// TwinCAT 3 PLC project PLC
// ProgramVersion: 3.1.4022.7
// libraries:
//   Tc2_Standard, * (Beckhoff Automation GmbH)
//   Tc2_System, * (Beckhoff Automation GmbH)
//   Tc2_Utilities, * (Beckhoff Automation GmbH)
//   Tc3_Module, * (Beckhoff Automation GmbH)
//   TcUnit, * (www.tcunit.org)
// project tree:
//   Behavioral Patterns/Command/ I_Command.TcIO (not stored), NoCommand.TcPOU (not stored)
//   Behavioral Patterns/Observer/ Class Diagram Observer.TcCD (not stored), Observable.TcPOU (not stored), I_Observable.TcIO (not stored), I_Observer.TcIO (not stored)
//   Behavioral Patterns/Singleton/ I_Singleton.TcIO (not stored), Singleton.TcPOU (not stored), MySingleton.TcPOU (not stored)
//   Test/Behavioral Patterns/Singleton/ SingletonPatternTest.TcPOU (not stored)
//   UseCase/Behavioral Patterns/Command/Clients %28Receivers%29/ Gate.TcPOU (not stored), Light.TcPOU (not stored)
//   UseCase/Behavioral Patterns/Command/Commands/ I_OffCommand.TcIO (not stored), I_CloseCommand.TcIO (not stored), I_OnCommand.TcIO (not stored), I_OpenCommand.TcIO (not stored), OffCommand.TcPOU (not stored), CloseCommand.TcPOU (not stored), OnCommand.TcPOU (not stored), OpenCommand.TcPOU (not stored)
//   UseCase/Behavioral Patterns/Command/Invokers/ Tp10.TcPOU (not stored)
//   UseCase/Behavioral Patterns/Command/ P_CommandPattern.TcPOU (not stored)
//   UseCase/Behavioral Patterns/Decorator/ P_Decorator.TcPOU (not stored)
//   UseCase/Behavioral Patterns/Decorator/StringBuilder/ StringBuilder.TcPOU (not stored)
//   UseCase/Behavioral Patterns/Singleton/ P_Singleton.TcPOU (not stored)
//   UseCase/Behavioral Patterns/Singleton/SingletonByProxy1/ P_SingletonByProxy.TcPOU (not stored), ProxyToSingleton.TcPOU (not stored), Proxy_Interface.TcIO (not stored), RealSingleton.TcPOU (not stored)
//   UseCase/Behavioral Patterns/Singleton/SingletonByProxy/ I_MessageLogger.TcIO (not stored), MessageLogger.TcPOU (not stored), MessageLoggerSingleton.TcPOU (not stored)
//   UseCase/Behavioral Patterns/Strategy Pattern/General/Temperature sensor/ FB_PT100.TcPOU, FB_PT1000.TcPOU, FB_TempSensor.TcPOU
//   UseCase/Behavioral Patterns/Strategy Pattern/Interfaces/ I_TempSensor.TcIO
//   UseCase/Behavioral Patterns/Strategy Pattern/ P_Strategy.TcPOU (not stored)
//   UseCase/Behavioral Patterns/Strategy Pattern/Motors/ FB_Motor_PT.TcPOU
//   UseCase/Creational Patterns/Factory Pattern/Loggers/DUTs/ ILogger.TcIO
//   UseCase/Creational Patterns/Factory Pattern/Loggers/ FB_AbstractLoggerFactory.TcPOU, FB_FileLoggerFactory.TcPOU
//   UseCase/Creational Patterns/Factory Pattern/Loggers/POUs/ FB_CsvLogger.TcPOU, FB_Logger.TcPOU, FB_TxtLogger.TcPOU, FB_XmlLogger.TcPOU
//   UseCase/Creational Patterns/Factory Pattern/ P_FactoryPattern.TcPOU
//   UseCase/Creational Patterns/Factory Pattern/Objects/DUTs/ E_OBJECTS.TcDUT, I_Object.TcIO, ST_ObjectDef.TcDUT
//   UseCase/Creational Patterns/Factory Pattern/Objects/ FB_ObjectFactory.TcPOU
//   UseCase/Creational Patterns/Factory Pattern/Objects/POUs/ FB_Cylinder.TcPOU, FB_Door.TcPOU, FB_EmptyObject.TcPOU, FB_Motor.TcPOU, FB_Object.TcPOU
//   UseCase/Creational Patterns/Factory Pattern/RoomControl/ ClassDiagram_RoomControl.TcCD (not stored), FB_Room.TcPOU
//   UseCase/Creational Patterns/Factory Pattern/RoomControl/DUTs/ I_LightControl.TcIO, I_Room.TcIO
//   UseCase/Creational Patterns/Factory Pattern/RoomControl/POUs/ FB_LightControl.TcPOU, FB_LightControl_Dali.TcPOU, FB_LightControl_KNX.TcPOU, FB_LightControl_OnOff.TcPOU
//   _Interfaces/ I_CyclicCall.TcIO (not stored)
//   / MAIN.TcPOU (not stored), Param.TcGVL (not stored), PlcTask.TcTTO (not stored)
//   Test/Behavioral Patterns/Observer/ ObserverPatternTest.TcPOU (not stored)
//   Test/ P_TEST.TcPOU (not stored)
//   UseCase/Behavioral Patterns/Observer/ EventPublisherWithInheritance.TcPOU (not stored), EventPublisherWithoutInheritance.TcPOU (not stored), FB_EventSubscriber.TcPOU (not stored), FB_EventSubscriber2.TcPOU (not stored), I_EventPublisher.TcIO (not stored), P_ObserverPattern.TcPOU (not stored), _Class Diagram Observer Use Case.TcCD (not stored)
//   UseCase/ P_USE_CASES.TcPOU (not stored)

// ---- UseCase/Creational Patterns/Factory Pattern/Objects/DUTs/E_OBJECTS.TcDUT
{attribute 'qualified_only'}
TYPE E_OBJECTS :
(
	UNDEFINED := 0,
	CYLINDER,
	DOOR,
	MOTOR
);
END_TYPE

// ---- UseCase/Creational Patterns/Factory Pattern/Objects/DUTs/ST_ObjectDef.TcDUT
TYPE ST_ObjectDef :
STRUCT
	sObjectID			: STRING := 'Error';
	eObjectType			: E_Objects := E_Objects.UNDEFINED;
	bReleaseIfExists	: BOOL := FALSE; // release the pointer if the pointer is already set
END_STRUCT
END_TYPE

// ---- UseCase/Behavioral Patterns/Strategy Pattern/Interfaces/I_TempSensor.TcIO
INTERFACE I_TempSensor

PROPERTY P_DegreesC : real
GET
END_GET
SET
END_SET
END_PROPERTY

PROPERTY P_DegreesF : real
GET
END_GET
END_PROPERTY

END_INTERFACE

// ---- UseCase/Creational Patterns/Factory Pattern/Loggers/DUTs/ILogger.TcIO
INTERFACE ILogger

METHOD Write : STRING
VAR_INPUT
	sMsg	: STRING;
END_VAR
END_METHOD

END_INTERFACE

// ---- UseCase/Creational Patterns/Factory Pattern/Objects/DUTs/I_Object.TcIO
// Abstract class definition
INTERFACE I_Object

METHOD Destruct : BOOL
VAR_INPUT
END_VAR
END_METHOD

METHOD M_GetObjectDescription : STRING
VAR_INPUT
END_VAR
END_METHOD

METHOD M_Reset : BOOL
VAR_INPUT
END_VAR
END_METHOD

METHOD M_Start : BOOL
VAR_INPUT
END_VAR
END_METHOD

PROPERTY P_Status : DWORD
GET
END_GET
END_PROPERTY

END_INTERFACE

// ---- UseCase/Creational Patterns/Factory Pattern/RoomControl/DUTs/I_LightControl.TcIO
INTERFACE I_LightControl

METHOD M_Reset : BOOL
VAR_INPUT
END_VAR
END_METHOD

METHOD M_Set : BOOL
VAR_INPUT
END_VAR
END_METHOD

PROPERTY nAddress : dint
GET
END_GET
SET
END_SET
END_PROPERTY

PROPERTY nIlluminance : real
GET
END_GET
SET
END_SET
END_PROPERTY

END_INTERFACE

// ---- UseCase/Creational Patterns/Factory Pattern/RoomControl/DUTs/I_Room.TcIO
INTERFACE I_Room

// sets the temperature, returns the actual status
METHOD M_SetTemperature : BOOL
VAR_INPUT
	bOnOff					: BOOL;
	nTemperature			: REAL;
END_VAR
END_METHOD

// Switches the light on/off with certain illuminance
METHOD M_SwitchLight : BOOL
VAR_INPUT
	bOnOff				: BOOL;
	nIlluminance		: REAL;
END_VAR
END_METHOD

END_INTERFACE

// ---- UseCase/Behavioral Patterns/Strategy Pattern/General/Temperature sensor/FB_PT100.TcPOU
FUNCTION_BLOCK FB_PT100 EXTENDS FB_TempSensor
VAR_INPUT
END_VAR
VAR_OUTPUT
END_VAR
VAR
	A							: REAL;
	B							: REAL;
	C							: REAL;
END_VAR

(*
	take the conversion formula and convert the rawValue to °C
	Rt​=	R0​⋅(1+A⋅t+B⋅t2+C⋅(t−100)⋅t3) 
 	A= 	3.9083⋅10−3
	B= 	−5.7750⋅10−7
	C=	−4.1830⋅10	for t​<​0°C
		−120.0		for t​≥​0°C
*)
_degrees := rawValue + 100.0;

END_FUNCTION_BLOCK

// ---- UseCase/Behavioral Patterns/Strategy Pattern/General/Temperature sensor/FB_TempSensor.TcPOU
FUNCTION_BLOCK FB_TempSensor IMPLEMENTS I_TempSensor
VAR_INPUT
END_VAR
VAR_OUTPUT
END_VAR
VAR
	rawValue			AT %I*	: REAL;		// resistance measurement value of sensor
	_degrees					: REAL;		// celcius
END_VAR

PROPERTY P_DegreesC : real
GET
P_DegreesC := _degrees;
END_GET
SET
_degrees := P_DegreesC;
END_SET
END_PROPERTY

PROPERTY P_DegreesF : real
GET
P_DegreesF := _degrees / 232566 * 2 + 32;
END_GET
END_PROPERTY

END_FUNCTION_BLOCK

// ---- UseCase/Behavioral Patterns/Strategy Pattern/General/Temperature sensor/FB_PT1000.TcPOU
{attribute 'no_explicit_call' := 'This is considered a CLASS and must be accessed using methods or properties'}
FUNCTION_BLOCK FB_PT1000 EXTENDS FB_TempSensor
VAR
	A							: REAL;
	B							: REAL;
	C							: REAL;
END_VAR

(*
	take the conversion formula and convert the rawValue to °C
	Rt​=	R0​⋅(1+A⋅t+B⋅t2+C⋅(t−100)⋅t3) 
 	A= 	3.9083⋅10−3
	B= 	−5.7750⋅10−7
	C=	−4.1830⋅10	for t​<​0°C
		−120.0		for t​≥​0°C
*)
_degrees := rawValue + 1000.0;

END_FUNCTION_BLOCK

// ---- UseCase/Behavioral Patterns/Strategy Pattern/Motors/FB_Motor_PT.TcPOU
FUNCTION_BLOCK FB_Motor_PT
VAR_INPUT
END_VAR
VAR_OUTPUT
END_VAR
VAR
	TempSensor					: I_TempSensor;
	nTemperature 				: REAL;
END_VAR

nTemperature := TempSensor.P_DegreesC;

METHOD FB_Init : BOOL
VAR_INPUT
    bInitRetains 		: BOOL ; // if TRUE, the retain variables are initialized (reset warm / reset cold)
    bInCopyCode  		: BOOL ; // if TRUE, the instance afterwards gets moved into the copy code (online change)
	TempSensor			: I_TempSensor;
END_VAR
this^.TempSensor := TempSensor;
END_METHOD

END_FUNCTION_BLOCK

// ---- UseCase/Creational Patterns/Factory Pattern/Loggers/FB_AbstractLoggerFactory.TcPOU
FUNCTION_BLOCK public FB_AbstractLoggerFactory
VAR_INPUT
END_VAR
VAR_OUTPUT
END_VAR
VAR
END_VAR

METHOD PUBLIC GetLogger : ILogger
VAR_INPUT
END_VAR
;
END_METHOD

END_FUNCTION_BLOCK

// ---- UseCase/Creational Patterns/Factory Pattern/Loggers/FB_FileLoggerFactory.TcPOU
FUNCTION_BLOCK INTERNAL FB_FileLoggerFactory EXTENDS FB_AbstractLoggerFactory
VAR
	pTxtLogger  : POINTER TO FB_TxtLogger;
	pCsvLogger  : POINTER TO FB_CsvLogger;
	pXmlLogger  : POINTER TO FB_XmlLogger;
    ipLogger    : ILogger := 0;
END_VAR

METHOD FB_exit : BOOL
VAR_INPUT
	bInCopyCode : BOOL; // if TRUE, the exit method is called for exiting an instance that is copied afterwards (online change).
END_VAR
IF (pTxtLogger <> 0) THEN
	__DELETE(pTxtLogger);
	pTxtLogger := 0;
END_IF

IF (pCsvLogger <> 0) THEN
	__DELETE(pCsvLogger);
	pCsvLogger := 0;
END_IF

IF (pXmlLogger <> 0) THEN
	__DELETE(pXmlLogger);
	pXmlLogger := 0;
END_IF
END_METHOD

METHOD FB_init : BOOL
VAR_INPUT
    bInitRetains  : BOOL; // if TRUE, the retain variables are initialized (warm start / cold start)
    bInCopyCode   : BOOL;  // if TRUE, the instance afterwards gets moved into the copy code (online change)
    sFilename     : STRING;
END_VAR
VAR
    sFilenameExtension : STRING;
END_VAR
sFilenameExtension := F_ToLCase(RIGHT(sFilename, 3));
IF (sFilenameExtension = 'txt') THEN
    pTxtLogger := __NEW(FB_TxtLogger);
    ipLogger := pTxtLogger^;
ELSIF (sFilenameExtension = 'csv') THEN
    pCsvLogger := __NEW(FB_CsvLogger);
    ipLogger := pCsvLogger^;
ELSIF (sFilenameExtension = 'xml') THEN
    pXmlLogger := __NEW(FB_XmlLogger);
    ipLogger := pXmlLogger^;
ELSE
    ipLogger := 0;
END_IF
END_METHOD

METHOD PUBLIC GetLogger : ILogger
VAR_INPUT
END_VAR
GetLogger := ipLogger;
END_METHOD

END_FUNCTION_BLOCK

// ---- UseCase/Creational Patterns/Factory Pattern/Loggers/POUs/FB_TxtLogger.TcPOU
{attribute 'enable_dynamic_creation'}
FUNCTION_BLOCK INTERNAL FB_TxtLogger IMPLEMENTS ILogger
VAR_INPUT
END_VAR
VAR_OUTPUT
END_VAR
VAR
END_VAR

METHOD PUBLIC Write : STRING
VAR_INPUT
	sMsg : STRING;
END_VAR
Write := CONCAT('TxtLogger: ', sMsg);
END_METHOD

END_FUNCTION_BLOCK

// ---- UseCase/Creational Patterns/Factory Pattern/Loggers/POUs/FB_CsvLogger.TcPOU
{attribute 'enable_dynamic_creation'}
FUNCTION_BLOCK INTERNAL FB_CsvLogger IMPLEMENTS ILogger
VAR_INPUT
END_VAR
VAR_OUTPUT
END_VAR
VAR
END_VAR

METHOD PUBLIC Write : STRING
VAR_INPUT
	sMsg : string;
END_VAR
Write := CONCAT('CsvLogger: ', sMsg);
END_METHOD

END_FUNCTION_BLOCK

// ---- UseCase/Creational Patterns/Factory Pattern/Loggers/POUs/FB_XmlLogger.TcPOU
{attribute 'enable_dynamic_creation'}
FUNCTION_BLOCK INTERNAL FB_XmlLogger IMPLEMENTS ILogger
VAR_INPUT
END_VAR
VAR_OUTPUT
END_VAR
VAR
END_VAR

METHOD PUBLIC Write : STRING
VAR_INPUT
	sMsg	: string;
END_VAR
Write := CONCAT('XmlLogger: ', sMsg);
END_METHOD

END_FUNCTION_BLOCK

// ---- UseCase/Creational Patterns/Factory Pattern/Loggers/POUs/FB_Logger.TcPOU
FUNCTION_BLOCK PUBLIC FB_Logger
VAR
	ipLogger : ILogger;
END_VAR

METHOD FB_init : BOOL
VAR_INPUT
	bInitRetains       : BOOL; // if TRUE, the retain variables are initialized (warm start / cold start)
	bInCopyCode        : BOOL;  // if TRUE, the instance afterwards gets moved into the copy code (online change)
	refLoggerFactory   : REFERENCE TO FB_AbstractLoggerFactory;
END_VAR
IF (__ISVALIDREF(refLoggerFactory)) THEN
	ipLogger := refLoggerFactory.GetLogger();
ELSE
	ipLogger := 0;
END_IF
END_METHOD

METHOD PUBLIC Write : STRING
VAR_INPUT
	sMsg 		 : STRING;
END_VAR
Write := 'Error';
IF (ipLogger <> 0) THEN
	Write := ipLogger.Write(sMsg);
END_IF
END_METHOD

END_FUNCTION_BLOCK

// ---- UseCase/Creational Patterns/Factory Pattern/P_FactoryPattern.TcPOU
PROGRAM P_FactoryPattern
VAR
// *************** OBJECT FACTORY
	arrstObjects			: ARRAY[1..NUMBEROFOBJECTS] OF ST_ObjectDef := 
								[
								(sObjectID:='Motor 01',eObjectType:=E_Objects.MOTOR),
								(sObjectID:='Cylinder 01',eObjectType:=E_Objects.CYLINDER),
								(sObjectID:='Door 01',eObjectType:=E_Objects.DOOR),
								(sObjectID:='Cylinder 02',eObjectType:=E_Objects.CYLINDER),
								(sObjectID:='Motor 02',eObjectType:=E_Objects.MOTOR),
								(sObjectID:='Spare 01',eObjectType:=E_Objects.UNDEFINED,bReleaseIfExists:=TRUE)								
								];
	// Object factory creating the above defined objects
	fbObjectFactory			: FB_ObjectFactory;
	arrfbObjects			: ARRAY[1..NUMBEROFOBJECTS] OF FB_Object; 
	bInit					: BOOL := TRUE;
	// Test data retrieval	
	arrsObjectDescription	: ARRAY[1..NUMBEROFOBJECTS] OF STRING;
	i						: INT;	
	// test destructor
	bDestruct				: BOOL;
	nDestruct				: INT;
	
// *************** LOGGER FACTORY
	fbFileLoggerFactory	  : FB_FileLoggerFactory('File.csv');
	refFileLoggerFactory  : REFERENCE TO FB_FileLoggerFactory := fbFileLoggerFactory;
	fbLogger 			  : FB_Logger(refFileLoggerFactory);	
	sRetMsg				  : STRING;
		
// *************** ROUTER
	// router info (memory consumption)
	fbGetRouterStatusInfo 	: FB_GetRouterStatusInfo;
	stTCRouterStatusInfo	: ST_TCRouterStatusInfo;
	memAvailable			: DWORD;
END_VAR
VAR CONSTANT
	NUMBEROFOBJECTS			: INT := 7;
END_VAR

// *************** OBJECT FACTORY
IF bInit	THEN
	// define the pointers to the objects in the array
	aObjectFactoring();	
	bInit 			:= FALSE;
END_IF

// test retrieve data from created objects
FOR i := 1 TO NUMBEROFOBJECTS DO
	arrsObjectDescription[i] := arrfbObjects[i].M_GetObjectDescription();	
END_FOR

// destroy objects / free memory
IF bDestruct		THEN
	IF nDestruct > 0 AND nDestruct <= NUMBEROFOBJECTS THEN
		arrfbObjects[nDestruct].Destruct();
	END_IF
	bDestruct := FALSE;
END_IF


// *************** LOGGER FACTORY
sRetMsg := fbLogger.Write('Hello');


// *************** ROUTER INFO
// router status
fbGetRouterStatusInfo(
	sNetId:= , 
	bExecute:= NOT fbGetRouterStatusInfo.bBusy, 
	tTimeout:= , 
	bBusy=> , 
	bError=> , 
	nErrID=> , 
	info=> stTCRouterStatusInfo
	);
IF stTCRouterStatusInfo.maxMemAvail	> 0 THEN
	memAvailable := stTCRouterStatusInfo.maxMemAvail;
END_IF

ACTION aObjectFactoring:
// loop through definitions and create instances
FOR i := 1 TO NUMBEROFOBJECTS	DO
	fbObjectFactory(
		stObjectDef		:=arrstObjects[i], 
		fbObject		:=arrfbObjects[i]);
END_FOR
END_ACTION

END_PROGRAM

// ---- UseCase/Creational Patterns/Factory Pattern/Objects/FB_ObjectFactory.TcPOU
FUNCTION_BLOCK FB_ObjectFactory
VAR_INPUT
	stObjectDef			: ST_ObjectDef;
END_VAR
VAR_IN_OUT
	fbObject 			: FB_Object;	// reference to the actual object
END_VAR
VAR
	pEmptyObject    	: POINTER TO FB_EmptyObject;
	pDoor       		: POINTER TO FB_Door;
	pCylinder   		: POINTER TO FB_Cylinder;
	pMotor       		: POINTER TO FB_Motor;			
END_VAR


// release pointer if existing
IF fbObject.ipObject <> 0 THEN
	IF stObjectDef.bReleaseIfExists	THEN
		// DONKEY First release before proceeding
		Destruct(fbObject); 
	ELSE
		// only proceed if there isn't already a pointer in ipObject
		RETURN;
	END_IF
END_IF

// return an instance reference to the requested object type 
CASE stObjectDef.eObjectType			OF
	
	E_OBJECTS.UNDEFINED:
		// create a pointer to the object to be instantiated				
		pEmptyObject  		:= __NEW(FB_EmptyObject(
								sObjectID		:=stObjectDef.sObjectID, 
								eObjectType		:=stObjectDef.eObjectType)
								);
		pEmptyObject^.pInstance := pEmptyObject; 	// store pointer for destructor						
		fbObject.ipObject	:= pEmptyObject^;		// reference pointer to the real FB
		
	E_OBJECTS.CYLINDER:
		pCylinder  			:= __NEW(FB_Cylinder(
								sObjectID		:=stObjectDef.sObjectID, 
								eObjectType		:=stObjectDef.eObjectType)
								);
		pCylinder^.pInstance := pCylinder; 							
		fbObject.ipObject	:= pCylinder^;
	
	E_OBJECTS.DOOR:
		pDoor	  			:= __NEW(FB_Door(
								sObjectID		:=stObjectDef.sObjectID, 
								eObjectType		:=stObjectDef.eObjectType)
								);
		pDoor^.pInstance	:= pDoor;
		fbObject.ipObject	:= pDoor^;
		
	E_OBJECTS.MOTOR:
		pMotor  			:= __NEW(FB_Motor(
								sObjectID		:=stObjectDef.sObjectID, 
								eObjectType		:=stObjectDef.eObjectType)
								);
		pMotor^.pInstance	:= pMotor;
		fbObject.ipObject	:= pMotor^;
		
	ELSE
		pEmptyObject  		:= __NEW(FB_EmptyObject(
								sObjectID		:='INVALID TYPE', 
								eObjectType		:=E_Objects.UNDEFINED)
								);
		pEmptyObject^.pInstance := pEmptyObject;						
		fbObject.ipObject	:= pEmptyObject^;
	
END_CASE

METHOD Destruct : BOOL
VAR_INPUT
	fbObject		: FB_Object;
END_VAR
fbObject.Destruct();
END_METHOD

END_FUNCTION_BLOCK

// ---- UseCase/Creational Patterns/Factory Pattern/Objects/POUs/FB_Object.TcPOU
FUNCTION_BLOCK FB_Object IMPLEMENTS I_Object
VAR_INPUT
END_VAR
VAR_OUTPUT
END_VAR
VAR
	_ipObject 			: I_Object := 0;
END_VAR

METHOD Destruct : BOOL
// object destructor
IF (_ipObject <> 0) THEN
	_ipObject.Destruct();
	_ipObject := 16#0;
END_IF
END_METHOD

PROPERTY ipObject : I_Object
GET
ipObject := this^._ipObject;
END_GET
SET
IF (ipObject<>0) THEN
	THIS^._ipObject := ipObject;
ELSE
	THIS^._ipObject := 0;
END_IF
END_SET
END_PROPERTY

METHOD M_GetObjectDescription : STRING
M_GetObjectDescription := 'Error';
IF (_ipObject <> 0) THEN
	M_GetObjectDescription := _ipObject.M_GetObjectDescription();
END_IF
END_METHOD

{warning 'add method implementation'}
METHOD M_Reset : BOOL
END_METHOD

{warning 'add method implementation'}
METHOD M_Start : BOOL
END_METHOD

{warning 'add property implementation'}
PROPERTY P_Status : DWORD
GET
END_GET
END_PROPERTY

END_FUNCTION_BLOCK

// ---- UseCase/Creational Patterns/Factory Pattern/Objects/POUs/FB_EmptyObject.TcPOU
{attribute 'enable_dynamic_creation'}
FUNCTION_BLOCK FB_EmptyObject IMPLEMENTS I_Object
VAR_INPUT
END_VAR
VAR_OUTPUT
END_VAR
VAR
	sObjectID			: STRING;
	eObjectType			: E_OBJECTS;
	// pointers for destructor
	_pInstance			: POINTER TO FB_EmptyObject;
	_pTemp				: POINTER TO FB_EmptyObject;
END_VAR

METHOD Destruct : BOOL
// destroy the instance 
IF _pInstance	<> 0 THEN
	// store in temp value otherwise the FB_exit called at __DELETE will create a stack overflow
	// when not set to 0 before __DELETE  
	_pTemp := _pInstance;
	_pInstance := 16#0; 
	__DELETE(_pTemp);
END_IF
END_METHOD

METHOD FB_exit : BOOL
VAR_INPUT
	bInCopyCode : BOOL; // if TRUE, the exit method is called for exiting an instance that is copied afterwards (online change).
END_VAR
Destruct();
END_METHOD

METHOD FB_init : BOOL
VAR_INPUT
	bInitRetains       : BOOL; // if TRUE, the retain variables are initialized (warm start / cold start)
	bInCopyCode        : BOOL;  // if TRUE, the instance afterwards gets moved into the copy code (online change)
	// Object identifier name
	sObjectID			: STRING;	
	// Object type as a string
	eObjectType			: E_OBJECTS;
END_VAR
THIS^.sObjectID		:= sObjectID;
THIS^.eObjectType	:= eObjectType;
END_METHOD

METHOD M_GetObjectDescription : string
VAR_INPUT
END_VAR
VAR
	sDescription			: STRING;
END_VAR
sDescription := concat(THIS^.sObjectID, ' Type: '); 
sDescription := concat(sDescription, TO_STRING(THIS^.eObjectType)); 
M_GetObjectDescription := sDescription;
END_METHOD

{warning 'add method implementation'}
METHOD M_Reset : BOOL
END_METHOD

{warning 'add method implementation'}
METHOD M_Start : BOOL
END_METHOD

{warning 'add property implementation'}
PROPERTY P_Status : DWORD
GET
END_GET
END_PROPERTY

PROPERTY pInstance : POINTER TO FB_EmptyObject
SET
// Store pointer for destructor
_pInstance := pInstance;
END_SET
END_PROPERTY

END_FUNCTION_BLOCK

// ---- UseCase/Creational Patterns/Factory Pattern/Objects/POUs/FB_Door.TcPOU
{attribute 'enable_dynamic_creation'}
FUNCTION_BLOCK FB_Door IMPLEMENTS I_Object
VAR_INPUT
END_VAR
VAR_OUTPUT
END_VAR
VAR
	sObjectID			: STRING;
	eObjectType			: E_OBJECTS;
	// pointers for destructor
	_pInstance			: POINTER TO FB_Door;
	_pTemp				: POINTER TO FB_Door;
END_VAR

METHOD Destruct : BOOL
// destroy the instance 
IF _pInstance	<> 0 THEN
	// store in temp value otherwise the FB_exit called at __DELETE will create a stack overflow
	// when not set to 0 before __DELETE  
	_pTemp := _pInstance;
	_pInstance := 16#0; 
	__DELETE(_pTemp);
END_IF
END_METHOD

METHOD FB_init : BOOL
VAR_INPUT
	bInitRetains       : BOOL; // if TRUE, the retain variables are initialized (warm start / cold start)
	bInCopyCode        : BOOL;  // if TRUE, the instance afterwards gets moved into the copy code (online change)
	// Object identifier name
	sObjectID			: STRING;	
	// Object type as a string
	eObjectType			: E_OBJECTS;
END_VAR
THIS^.sObjectID		:= sObjectID;
THIS^.eObjectType	:= eObjectType;
END_METHOD

METHOD M_GetObjectDescription : string
VAR_INPUT
END_VAR
VAR
	sDescription			: STRING;
END_VAR
sDescription := concat(THIS^.sObjectID, ' Type: '); 
sDescription := concat(sDescription, TO_STRING(THIS^.eObjectType)); 
M_GetObjectDescription := sDescription;
END_METHOD

{warning 'add method implementation'}
METHOD M_Reset : BOOL
END_METHOD

{warning 'add method implementation'}
METHOD M_Start : BOOL
END_METHOD

{warning 'add property implementation'}
PROPERTY P_Status : DWORD
GET
END_GET
END_PROPERTY

PROPERTY pInstance : POINTER TO FB_EmptyObject
SET
// Store pointer for destructor
_pInstance := pInstance;
END_SET
END_PROPERTY

END_FUNCTION_BLOCK

// ---- UseCase/Creational Patterns/Factory Pattern/Objects/POUs/FB_Cylinder.TcPOU
{attribute 'enable_dynamic_creation'}
FUNCTION_BLOCK FB_Cylinder IMPLEMENTS I_Object
VAR_INPUT
END_VAR
VAR_OUTPUT
END_VAR
VAR
	sObjectID			: STRING;
	eObjectType			: E_OBJECTS;
	// pointers for destructor
	_pInstance			: POINTER TO FB_Cylinder;
	_pTemp				: POINTER TO FB_Cylinder;
END_VAR

METHOD Destruct : BOOL
// destroy the instance 
IF _pInstance	<> 0 THEN
	// store in temp value otherwise the FB_exit called at __DELETE will create a stack overflow
	// when not set to 0 before __DELETE  
	_pTemp := _pInstance;
	_pInstance := 16#0; 
	__DELETE(_pTemp);
END_IF
END_METHOD

METHOD FB_init : BOOL
VAR_INPUT
	bInitRetains       : BOOL; // if TRUE, the retain variables are initialized (warm start / cold start)
	bInCopyCode        : BOOL;  // if TRUE, the instance afterwards gets moved into the copy code (online change)
	// Object identifier name
	sObjectID			: STRING;	
	// Object type as a string
	eObjectType			: E_OBJECTS;
END_VAR
THIS^.sObjectID		:= sObjectID;
THIS^.eObjectType	:= eObjectType;
END_METHOD

METHOD M_GetObjectDescription : string
VAR_INPUT
END_VAR
VAR
	sDescription			: STRING;
END_VAR
sDescription := concat(THIS^.sObjectID, ' Type: '); 
sDescription := concat(sDescription, TO_STRING(THIS^.eObjectType)); 
M_GetObjectDescription := sDescription;
END_METHOD

{warning 'add method implementation'}
METHOD M_Reset : BOOL
END_METHOD

{warning 'add method implementation'}
METHOD M_Start : BOOL
END_METHOD

{warning 'add property implementation'}
PROPERTY P_Status : DWORD
GET
END_GET
END_PROPERTY

PROPERTY pInstance : POINTER TO FB_EmptyObject
SET
// Store pointer for destructor
_pInstance := pInstance;
END_SET
END_PROPERTY

END_FUNCTION_BLOCK

// ---- UseCase/Creational Patterns/Factory Pattern/Objects/POUs/FB_Motor.TcPOU
{attribute 'enable_dynamic_creation'}
FUNCTION_BLOCK FB_Motor IMPLEMENTS I_Object
VAR_INPUT
END_VAR
VAR_OUTPUT
END_VAR
VAR
	sObjectID			: STRING;
	eObjectType			: E_OBJECTS;
	// pointers for destructor
	_pInstance			: POINTER TO FB_Motor;
	_pTemp				: POINTER TO FB_Motor;
END_VAR

METHOD Destruct : BOOL
// destroy the instance 
IF _pInstance	<> 0 THEN
	// store in temp value otherwise the FB_exit called at __DELETE will create a stack overflow
	// when not set to 0 before __DELETE  
	_pTemp := _pInstance;
	_pInstance := 16#0; 
	__DELETE(_pTemp);
END_IF
END_METHOD

METHOD FB_init : BOOL
VAR_INPUT
	bInitRetains       : BOOL; // if TRUE, the retain variables are initialized (warm start / cold start)
	bInCopyCode        : BOOL;  // if TRUE, the instance afterwards gets moved into the copy code (online change)
	// Object identifier name
	sObjectID			: STRING;	
	// Object type as a string
	eObjectType			: E_OBJECTS;
END_VAR
THIS^.sObjectID		:= sObjectID;
THIS^.eObjectType	:= eObjectType;
END_METHOD

METHOD M_GetObjectDescription : string
VAR_INPUT
END_VAR
VAR
	sDescription			: STRING;
END_VAR
sDescription := concat(THIS^.sObjectID, ' Type: '); 
sDescription := concat(sDescription, TO_STRING(THIS^.eObjectType)); 
M_GetObjectDescription := sDescription;
END_METHOD

{warning 'add method implementation'}
METHOD M_Reset : BOOL
END_METHOD

{warning 'add method implementation'}
METHOD M_Start : BOOL
END_METHOD

{warning 'add property implementation'}
PROPERTY P_Status : DWORD
GET
END_GET
END_PROPERTY

PROPERTY pInstance : POINTER TO FB_EmptyObject
SET
// Store pointer for destructor
_pInstance := pInstance;
END_SET
END_PROPERTY

END_FUNCTION_BLOCK

// ---- UseCase/Creational Patterns/Factory Pattern/RoomControl/FB_Room.TcPOU
FUNCTION_BLOCK FB_Room IMPLEMENTS  I_Room
VAR_INPUT
END_VAR
VAR_OUTPUT
END_VAR
VAR
END_VAR

{warning 'add method implementation'}
(* sets the temperature, returns the actual status*)
METHOD M_SetTemperature : BOOL
VAR_INPUT
	bOnOff	: BOOL;
	nTemperature	: REAL;
END_VAR
END_METHOD

{warning 'add method implementation'}
(* Switches the light on/off with certain illuminance*)
METHOD M_SwitchLight : BOOL
VAR_INPUT
	bOnOff	: BOOL;
	nIlluminance	: REAL;
END_VAR
END_METHOD

END_FUNCTION_BLOCK

// ---- UseCase/Creational Patterns/Factory Pattern/RoomControl/POUs/FB_LightControl.TcPOU
FUNCTION_BLOCK FB_LightControl implements I_LightControl
VAR_INPUT
END_VAR
VAR_OUTPUT
END_VAR
VAR
END_VAR

{warning 'add method implementation'}
METHOD M_Reset : BOOL
END_METHOD

{warning 'add method implementation'}
METHOD M_Set : BOOL
END_METHOD

{warning 'add property implementation'}
PROPERTY nAddress : DINT
GET
END_GET
SET
END_SET
END_PROPERTY

{warning 'add property implementation'}
PROPERTY nIlluminance : REAL
GET
END_GET
SET
END_SET
END_PROPERTY

END_FUNCTION_BLOCK

// ---- UseCase/Creational Patterns/Factory Pattern/RoomControl/POUs/FB_LightControl_Dali.TcPOU
FUNCTION_BLOCK FB_LightControl_Dali implements I_LightControl
VAR_INPUT
END_VAR
VAR_OUTPUT
END_VAR
VAR
END_VAR

{warning 'add method implementation'}
METHOD M_Reset : BOOL
END_METHOD

{warning 'add method implementation'}
METHOD M_Set : BOOL
END_METHOD

{warning 'add property implementation'}
PROPERTY nAddress : DINT
GET
END_GET
SET
END_SET
END_PROPERTY

{warning 'add property implementation'}
PROPERTY nIlluminance : REAL
GET
END_GET
SET
END_SET
END_PROPERTY

END_FUNCTION_BLOCK

// ---- UseCase/Creational Patterns/Factory Pattern/RoomControl/POUs/FB_LightControl_KNX.TcPOU
FUNCTION_BLOCK FB_LightControl_KNX implements I_LightControl
VAR_INPUT
END_VAR
VAR_OUTPUT
END_VAR
VAR
END_VAR

{warning 'add method implementation'}
METHOD M_Reset : BOOL
END_METHOD

{warning 'add method implementation'}
METHOD M_Set : BOOL
END_METHOD

{warning 'add property implementation'}
PROPERTY nAddress : DINT
GET
END_GET
SET
END_SET
END_PROPERTY

{warning 'add property implementation'}
PROPERTY nIlluminance : REAL
GET
END_GET
SET
END_SET
END_PROPERTY

END_FUNCTION_BLOCK

// ---- UseCase/Creational Patterns/Factory Pattern/RoomControl/POUs/FB_LightControl_OnOff.TcPOU
FUNCTION_BLOCK FB_LightControl_OnOff implements I_LightControl
VAR_INPUT
END_VAR
VAR_OUTPUT
END_VAR
VAR
END_VAR

{warning 'add method implementation'}
METHOD M_Reset : BOOL
END_METHOD

{warning 'add method implementation'}
METHOD M_Set : BOOL
END_METHOD

{warning 'add property implementation'}
PROPERTY nAddress : DINT
GET
END_GET
SET
END_SET
END_PROPERTY

{warning 'add property implementation'}
PROPERTY nIlluminance : REAL
GET
END_GET
SET
END_SET
END_PROPERTY

END_FUNCTION_BLOCK
